ABB RobotStudio station: test1215.rspag

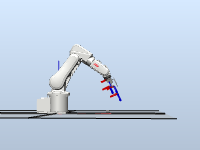
--- station ---
Station Solution7 (saved by RobotStudio 6.5.7392.129)
Controller System1
  mechanical unit ROB_1: IRB120_3_58__01, 6 joints, base frame (0, 0, 0) mm
Layout (positions relative to the parent item):
  - IRB120_3_58__01 [mechanism, from Robots\IRB120_3_58_G_01.rslib] at (0, 0, 0) mm; joint values [0, 0.627, 0, 0, 0.5236, 0] (rad or m)
  - SmartComponent_1 [smart component] at (473.41, 0, 322.42) mm, rotated rx 180 ry 24.08 rz 180 deg
      signals: DI GET, DO FINISH
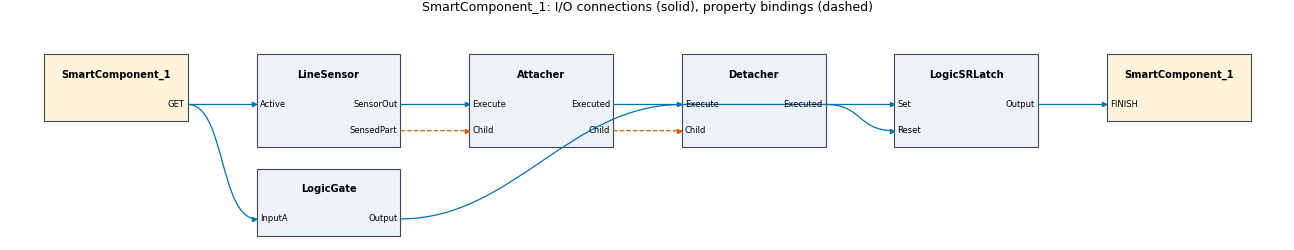
      connections:
        SmartComponent_1.GET -> LineSensor.Active
        SmartComponent_1.GET -> LogicGate.InputA
        LineSensor.SensorOut -> Attacher.Execute
        LogicGate.Output -> Detacher.Execute
        Attacher.Executed -> LogicSRLatch.Set
        Detacher.Executed -> LogicSRLatch.Reset
        LogicSRLatch.Output -> SmartComponent_1.FINISH
        LineSensor.SensedPart => Attacher.Child
        Attacher.Child => Detacher.Child
    - My_Mechanism  [mechanism] at (0, 0, 0) mm; joint values [0.01] (rad or m)
        TCP tool1 at (15.5, 0, 69.3) mm
        TCP tool2 at (-22.5, 0, 83.55) mm
        TCP tool3 at (-22.5, 0, 160.55) mm
        links: L1, L2
    - LineSensor [smart component, from Components\LineSensor.rslib] at (-22.5, 0, 81.55) mm
        properties: Start=[0 0 0]; End=[0 0 0.0125]; Radius=0.005; SensedPart=部件_1; SensedPoint=[0.465018035888672 -1.91242074260023E-15 0.0325653190612793]
      - _sensorPart_ [part]
    - Attacher [smart component, from Components\Attacher.rslib]
        properties: Parent=SmartComponent_1; Flange=0; Child=部件_1; Mount=false; Offset=[0 0 0]; Orientation=[0 0 0]
    - Detacher [smart component, from Components\Detacher.rslib]
        properties: Child=部件_1; KeepPosition=true
    - LogicGate [smart component, from Components\LogicGate.rslib]
        properties: Operator=NOT; Delay=0
    - LogicSRLatch [smart component, from Components\LogicSRLatch.rslib]
  - 部件_1 [part] at (1.09, 0, 0) mm, rotated rx 0 ry -0.22 rz 0 deg
  - 框架_1 [frame] at (15.5, 0, 69.3) mm
  - 框架_2 [frame] at (-22.5, 0, 83.55) mm
  - 框架_3 [frame] at (-22.5, 0, 160.55) mm
Attachment: SmartComponent_1 is attached to IRB120_3_58__01 / Link6
EventTableEntry 997: Group=, Trigger=DO_007 998, Actions=[EventTableActionMechanicalPose 999], Comment=, ActivationMode=2, Cyclic=false
EventTableTriggerIO 998: IOValue=[1], IRC5Controller=? -1, Operator=0, SignalSource=System1 498
EventTableActionMechanicalPose 999: VirtualSignal=, Mechanism=My_Mechanism  983, ToPoseName=SyncPosition, VirtualSignalValue=[1]
EventTableEntry 1000: Group=, Trigger=DO_007 1001, Actions=[EventTableActionMechanicalPose 1002], Comment=, ActivationMode=2, Cyclic=false
EventTableTriggerIO 1001: IOValue=[0], IRC5Controller=? -1, Operator=0, SignalSource=System1 498
EventTableActionMechanicalPose 1002: VirtualSignal=, Mechanism=My_Mechanism  983, ToPoseName=HomePosition, VirtualSignalValue=[1]
Station logic (signal -> signal, property => property):
  System1.DO_007 -> SmartComponent_1.GET
Targets, tools, work objects and paths stored in the station and not in the controller backup, written as RAPID:
! task T_ROB1
MODULE CalibData
  PERS tooldata tool1:=[TRUE,[[15.5,0,69.3],[1,0,0,0]],[1,[0,0,1],[1,0,0,0],0,0,0]];
  PERS tooldata tool2:=[TRUE,[[-22.5,0,83.55],[1,0,0,0]],[1,[0,0,1],[1,0,0,0],0,0,0]];
  PERS tooldata tool3:=[TRUE,[[-22.5,0,160.55],[1,0,0,0]],[1,[0,0,1],[1,0,0,0],0,0,0]];
ENDMODULE


--- Backups/System1/RAPID/TASK1/PROGMOD/MainModule.mod ---
MODULE MainModule
    !***********************************************************
    !
    ! 模块：$$未扩展的文件名$$
    !
    ! 描述:
    !   <在此处插入描述>
    !
    ! 作者: $$用户名$$
    !
    ! 版本: 1.0
    !
    !***********************************************************


    !***********************************************************
    !
    ! 主要程序
    !
    !   此处为程序入口点
    !
    !***********************************************************
    PROC main()
        !在此处添加代码
    ENDPROC
ENDMODULE

--- Backups/System1/RAPID/TASK1/SYSMOD/LINKEDM.sys ---
%%%
  VERSION:1
  LANGUAGE:ENGLISH
%%%

MODULE LINKEDM (SYSMODULE)

! FOLLOWER
!     Name of electronically linked follower axis used by operator at teach pendent.
      PERS string l_f_axis_name{5}       :=  ["",  "", "", "", ""];

!     Name of the mechanical unit for follower axis.
      PERS string l_f_mecunt_n{5}  :=  ["", "", "", "", ""];

!     Linked follower axis number in the mechanical unit (first axis in mech. unit is number 1).
      PERS num l_f_axis_no{5}      :=  [0,          0,   0,  0,  0];

! MASTER
!     Name of the mechanical unit for linked master axis.
      PERS string l_m_mecunt_n{5} :=  ["", "", "", "", ""];

!     Linked master axis number in the mechanical unit (first axis in mech. unit is number 1).
!     See axis number table in documentation for different master mechanical units.
      PERS num l_m_axis_no{5}     :=  [0,  0,  0,  0,  0];

! POSITION OFFSET
!     The increase of the allowed offset position between the master and follower
!     positions, used when starting AUTO mode. As soon as the offset is decreased
!     the old configurated parameter is used.
!     Example: 3 => the configurated value of allowed offset is increased 3 times.
      PERS num offset_ratio{5}       :=  [10,  10,   10,  10,  10];

! SPEED RATIO
!     Speed_ratio used in AUTO and JOG modes [ very_slow   slow    normal    fast]
!     Value 1 = max allowed manual speed.
      CONST num speed_ratio {20}      := [0.01, 0.01, 0.01, 0.01, 0.01,
                                          0.05, 0.05, 0.05, 0.05, 0.05,
                                          0.20, 0.20, 0.20, 0.20, 0.20,
                                          1.00, 1.00, 1.00, 1.00, 1.00];

! STEP SIZE
!     Displacement position used in JOG mode for each activation of positive or
!     negative movement.                  [very_short    short   normal   long]
!     Unit degees or meter.
      CONST num displacement {20}     := [0.001, 0.001, 0.001, 0.001, 0.001,
                                          0.005, 0.005, 0.005, 0.005, 0.005,
                                          0.020, 0.020, 0.020, 0.020, 0.020,
                                          0.100, 0.100, 0.100, 0.100, 0.100];


!-------------------------------------------------------------
 PROC Linked_m ()
      Linked_m_exe ;
 ENDPROC
ENDMODULE

--- Backups/System1/SYSPAR/EIO.cfg ---
EIO:CFG_1.0:6:1::
#
INDUSTRIAL_NETWORK:

      -Name "DeviceNet" -Label "DeviceNet Master/Slave Network" -Address "2"
#
DEVICENET_DEVICE:

      -Name "d652" -VendorName "ABB Robotics" -ProductName "24 VDC I/O Device"\
      -Label "DSQC 652 24 VDC I/O Device" -Address 10 -ProductCode 26\
      -DeviceType 7 -ConnectionType "COS" -OutputSize 2 -InputSize 2
#
DEVICENET_INTERNAL_DEVICE:

      -Name "DN_Internal_Device" -VendorName "ABB Robotics"\
      -ProductName "DeviceNet Internal Slave Device"
#
EIO_SIGNAL:

      -Name "DO_007" -SignalType "DO" -Device "d652" -DeviceMap "7"
